PROGRAM SafetyHandling
VAR
	// power on delay
	start_delay 	: TON := (PT := T#2S);
	// pulse for error acknowledgement
	ErrAck_Pulse	: TP := (PT := T#500MS);
	// pulse for safety restart
	restart_pulse 	: TP := (PT := T#500MS);
	// trigger for falling edge of error acknowledgement
	ErrAck_Trigger	: F_TRIG;
	// Errack logging
	ErrAckLog		: FB_EventLog;
	// restart logging
	RestartLog		: FB_EventLog;
	// safety logging
	SafetyLog		: FB_EventLog;
	
END_VAR
VAR_OUTPUT
	// error condition
	Error			: BOOL;
	// Emergency_stop engaged
	Emergency_stop	: BOOL;
END_VAR
VAR_INPUT
	// issue a remote restart
	remote_restart:		BOOL;
	// issue a remote Error Acknowledgment
	remote_ErrAck:		BOOL;
	// issue a remute run/stop
	remote_run:			BOOL := TRUE;
END_VAR

// Safety aus running on start
GVL_Safety.Run := remote_run;
// power on delay for Safety RESTART after RUN=1

// wait n seconds after Start ...
start_delay(IN := TRUE);
// ... and send ErrAck for n milliseconds
ErrAck_Pulse(IN := (GVL_Safety.State = 2) AND start_delay.Q);

// Error Acknowledgment: Turn key_switch OFF and press STOP 
GVL_Safety.ErrAck := (GVL_Main.key_switch_remote AND GVL_Main.reset_switch)
					OR ErrAck_Pulse.Q;
					//OR remote_ErrAck;
// detect falling edge 
//ErrAck_Trigger(CLK := GVL_Safety.ErrAck);
// send restart pulse on falling edge of ErrAck
//restart_pulse(IN := ErrAck_Trigger.Q);

// RESTART Safety after pushing reset or power on delay
GVL_Safety.Restart := (GVL_Main.key_switch_remote AND GVL_Main.start_switch)
 					   OR remote_restart;
        //               OR restart_pulse.Q;
				
//Error := GVL_Safety.Error OR (GVL_Safety.State <> 1);

//Emergency_stop := NOT GVL_Safety.Stop;

ErrAckLog(	Trigger := GVL_Safety.ErrAck,
			OnMessage := 'Safety error was acknowledged.');
			
RestartLog(	Trigger := GVL_Safety.Restart,
			Level := ADSLOG_MSGTYPE_WARN,
			OnMessage := 'Safety was restarted.');

SafetyLog(	Trigger := Error,
			Level := ADSLOG_MSGTYPE_ERROR,
			OnMessage := 'Safety Error! Emergency stop enganged!',
			OffMessage := 'Safety is OK.',
			OffLevel := ADSLOG_MSGTYPE_HINT);

END_PROGRAM

(* stored: Version 1.1.0.1, ProductVersion 3.1.4024.12
   POU SafetyHandling: Id {6d4a788c-2168-4769-93de-c67314036861}, SpecialFunc None *)
